TYPE T_ISO8601Time : STRING(30);
END_TYPE

(* stored: Version 1.1.0.1
   DUT T_ISO8601Time: Id {484f3032-af4f-4df9-99a0-ffc3fade2bb1} *)
